INTERFACE I_ExtensionVisitor

METHOD VisitExtension
VAR_INPUT
	VisitingExtension : I_Extension;
END_VAR
END_METHOD

END_INTERFACE

(* stored: Version 1.1.0.1, ProductVersion 3.1.4024.12
   Itf I_ExtensionVisitor: Id {8721962a-1337-07f3-0925-db9e62f9d4cc}
   Method VisitExtension: Id {04c103fa-d034-0249-09c2-8a238d2f5ab6} *)
